Staubli VAL3: onInsert.pgx

public program onInsert(string& x_sItem[])
  local string l_sEvent
  local num l_nKey
  local num l_nIndex
  local num l_nSize
  local num i
begin
  // get the traj type
end
